(* Schneider Machine Expert - Basic project SHREDDER, file version 2.8.0.0 *)
(* ProjectInformations: Name=Mulino Bazzica *)
(* UserInformations: LastName=Dominici, FirstName=Erica, PhoneNumber=+39 0742 38501, Email=info@promas.com, Street=via XXV Aprile, 10/12, City=Trevi, ZipCode=06039, State=Perugia, Country=Italy *)

HARDWARE
  Cpu 0: TM221CE16T
  EthernetConfiguration: NetworkName=M221, IpAllocationMode=FixedAddress, IpAddress=192.168.0.230, SubnetMask=255.255.254.0
  SerialLineConfiguration: Baud=Baud19200, Parity=ParityEven, DataBits=DataBits8, StopBits=StopBits1, PhysicalMedium=PhysicalMediumRs485, TransmissionMode=TransmissionModeModbusRtu, SlaveId=1, Addressing=SlaveAddressing
  MastTask: UsePeriodScanMode=true, PeriodScan=100
  FastTask: Period=255
  CpuBehavior: StartingMode=StartInRun, AutoSaveRamOnEeprom=true, WatchdogPeriod=250

SYMBOLS  (address, symbol, comment, settings)
  %M0       KM_ALL_ON
  %M1       KM_M1_ON
  %M2       ALARM_KM1
  %M3       ALARM_QM1
  %M4       ALARM_EXTERNAL
  %MW0      FSM_RECYCLING
  %MW4      ALARMS
  %MW6      HMI_INP  "PLC INPUT STATUS"
  %MW7      HMI_OUT  "PLC OUTPUT STATUS"
  %MW8      HMI_CMD  "PLC COMMANDS"
  %MW10     MACHINE_STATE
  %MW18     BLOWER_TIME  "O0 - BLOWER ON"
  %MW19     BLOWER_DELAY_OFF  "O0 - BLOWER DELAY OFF TIME"
  %MW20     VALVES_TIME  "O1-VALVES_SWITCH"
  %TM0      TON_VALVES  [Base=OneSecond, IsDynamicPreset=true]
  %TM1      TON_M1  [Preset=10, Base=OneSecond, IsDynamicPreset=true]
  %TM2      M1_ALM_ON  [Preset=3, Base=OneSecond]
  %TM3      M1_ALM_OFF  [Preset=3, Base=OneSecond]
  %TM4      QM1_ALM_ON  [Preset=3, Base=OneSecond]
  %TM5      QM1_ALM_OFF  [Preset=3, Base=OneSecond]
  %TM6      TON_M1_OFF  [Preset=3, IsDynamicPreset=true]
  %TM7      MULINO_ALM_ON  [Preset=3, Base=OneSecond]
  %TM8      MULINO_ALM_OFF  [Preset=3, Base=OneSecond]
  %I0.0     FDBK_TERMICO_QM1  "MGNETOTERMICO QM1"
  %I0.1     CONTATTORE_KM1  "CONTATTORE KM1"
  %I0.2     START_BTN  "START"
  %I0.3     STOP_BTN  "STOP"
  %I0.4     GENERAL_ERR_MULINO  "ERRORE MULINO"
  %Q0.0     VALVE1_2  "VALVES 12"
  %Q0.1     SILO_2_P  "SOLO PICCOLO"
  %Q0.2     SILO_1_G  "SILO GRANDE"
  %Q0.6     CONTACTOR_ON  "FAN"

POU IN
  (* SectionNumber=1 *)

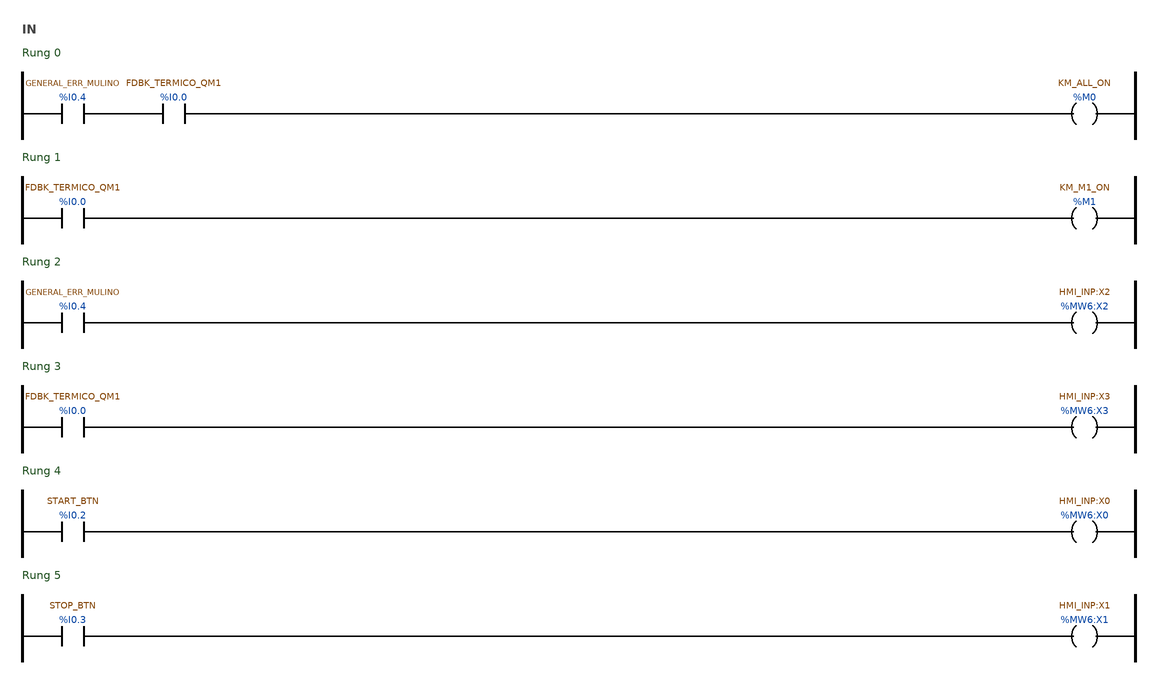

// Rung 0
  LD %I0.4                (* GENERAL_ERR_MULINO *)
  AND %I0.0               (* FDBK_TERMICO_QM1 *)
  ST %M0                  (* KM_ALL_ON *)
  // as ST:
  //   KM_ALL_ON := GENERAL_ERR_MULINO AND FDBK_TERMICO_QM1;

// Rung 1
  LD %I0.0                (* FDBK_TERMICO_QM1 *)
  ST %M1                  (* KM_M1_ON *)
  // as ST:
  //   KM_M1_ON := FDBK_TERMICO_QM1;

// Rung 2
  LD %I0.4                (* GENERAL_ERR_MULINO *)
  ST %MW6:X2              (* HMI_INP *)
  // as ST:
  //   HMI_INP:X2 := GENERAL_ERR_MULINO;

// Rung 3
  LD %I0.0                (* FDBK_TERMICO_QM1 *)
  ST %MW6:X3              (* HMI_INP *)
  // as ST:
  //   HMI_INP:X3 := FDBK_TERMICO_QM1;

// Rung 4
  LD %I0.2                (* START_BTN *)
  ST %MW6:X0              (* HMI_INP *)
  // as ST:
  //   HMI_INP:X0 := START_BTN;

// Rung 5
  LD %I0.3                (* STOP_BTN *)
  ST %MW6:X1              (* HMI_INP *)
  // as ST:
  //   HMI_INP:X1 := STOP_BTN;

POU FSM
  (* SectionNumber=2 *)

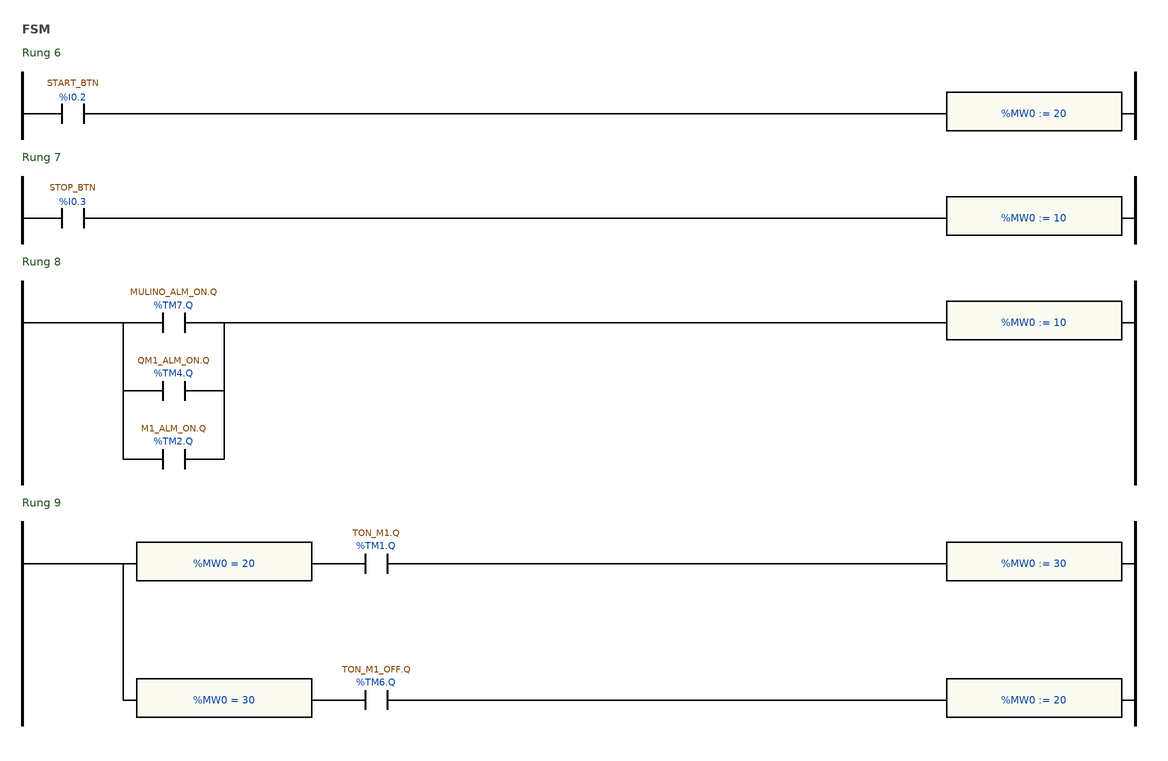

// Rung 6
  LD %I0.2                (* START_BTN *)
  [ %MW0 := 20 ]          (* FSM_RECYCLING *)
  // as ST:
  //   IF START_BTN THEN FSM_RECYCLING := 20; END_IF;

// Rung 7
  LD %I0.3                (* STOP_BTN *)
  [ %MW0 := 10 ]          (* FSM_RECYCLING *)
  // as ST:
  //   IF STOP_BTN THEN FSM_RECYCLING := 10; END_IF;

// Rung 8
  LD 1
  AND( %TM7.Q             (* MULINO_ALM_ON *)
  OR %TM4.Q               (* QM1_ALM_ON *)
  OR %TM2.Q               (* M1_ALM_ON *)
  )
  [ %MW0 := 10 ]          (* FSM_RECYCLING *)
  // as ST:
  //   IF MULINO_ALM_ON.Q OR QM1_ALM_ON.Q OR M1_ALM_ON.Q THEN FSM_RECYCLING := 10; END_IF;

// Rung 9
  LD 1
  MPS
  AND [ %MW0 = 20 ]       (* FSM_RECYCLING *)
  AND %TM1.Q              (* TON_M1 *)
  [ %MW0 := 30 ]          (* FSM_RECYCLING *)
  MPP
  AND [ %MW0 = 30 ]       (* FSM_RECYCLING *)
  AND %TM6.Q              (* TON_M1_OFF *)
  [ %MW0 := 20 ]          (* FSM_RECYCLING *)
  // as ST:
  //   IF FSM_RECYCLING = 20 AND TON_M1.Q THEN FSM_RECYCLING := 30; END_IF;
  //   IF FSM_RECYCLING = 30 AND TON_M1_OFF.Q THEN FSM_RECYCLING := 20; END_IF;

POU TIMERS
  (* SectionNumber=3 *)

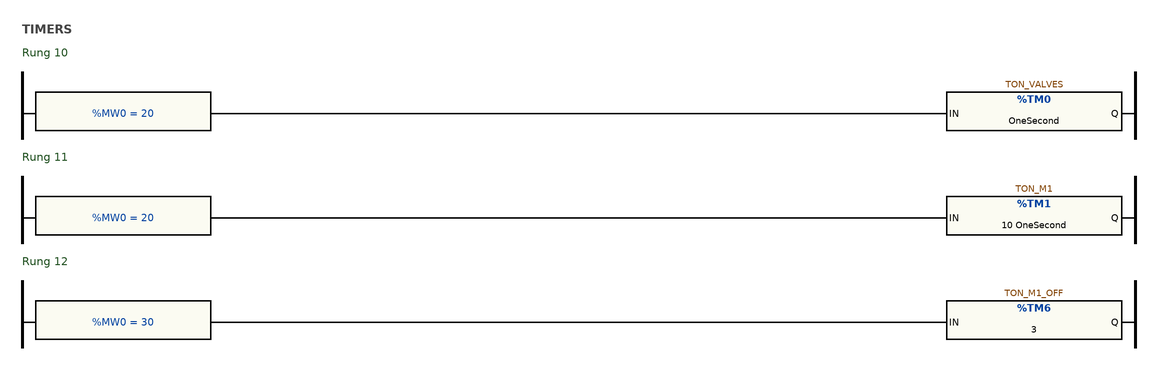

// Rung 10
  BLK %TM0                (* TON_VALVES *)
  LD [ %MW0 = 20 ]        (* FSM_RECYCLING *)
  IN
  END_BLK
  // as ST:
  //   TON_VALVES(IN := FSM_RECYCLING = 20);

// Rung 11
  BLK %TM1                (* TON_M1 *)
  LD [ %MW0 = 20 ]        (* FSM_RECYCLING *)
  IN
  END_BLK
  // as ST:
  //   TON_M1(IN := FSM_RECYCLING = 20);

// Rung 12
  BLK %TM6                (* TON_M1_OFF *)
  LD [ %MW0 = 30 ]        (* FSM_RECYCLING *)
  IN
  END_BLK
  // as ST:
  //   TON_M1_OFF(IN := FSM_RECYCLING = 30);

POU OUT
  (* SectionNumber=4 *)

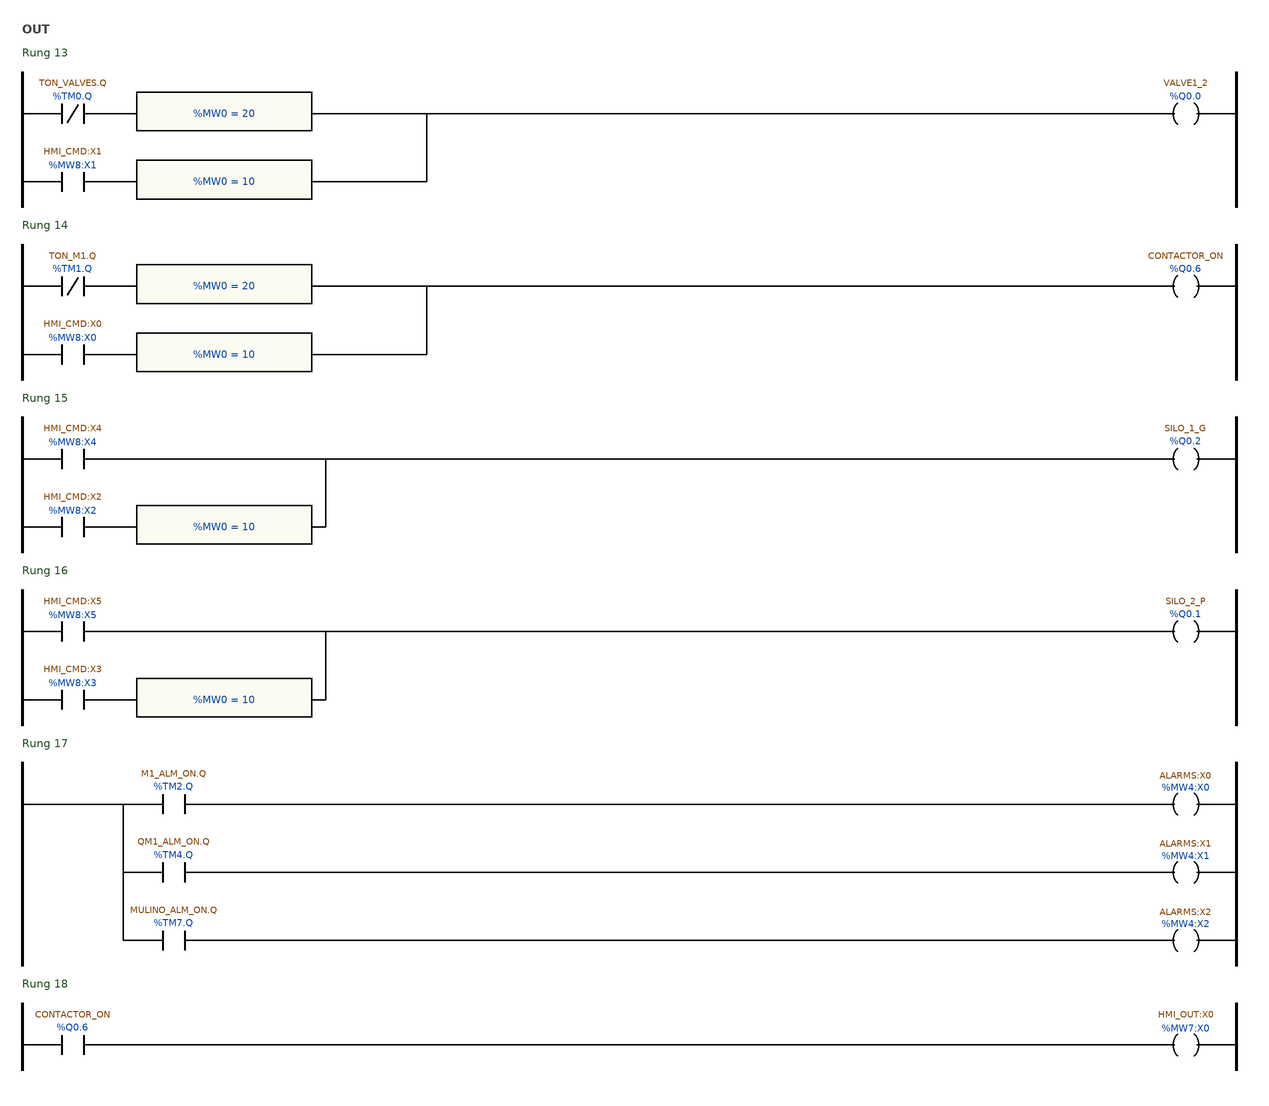

// Rung 13
  LDN %TM0.Q              (* TON_VALVES *)
  AND [ %MW0 = 20 ]       (* FSM_RECYCLING *)
  OR( %MW8:X1             (* HMI_CMD *)
  AND [ %MW0 = 10 ]       (* FSM_RECYCLING *)
  )
  ST %Q0.0                (* VALVE1_2 *)
  // as ST:
  //   VALVE1_2 := NOT TON_VALVES.Q AND FSM_RECYCLING = 20 OR HMI_CMD:X1 AND FSM_RECYCLING = 10;

// Rung 14
  LDN %TM1.Q              (* TON_M1 *)
  AND [ %MW0 = 20 ]       (* FSM_RECYCLING *)
  OR( %MW8:X0             (* HMI_CMD *)
  AND [ %MW0 = 10 ]       (* FSM_RECYCLING *)
  )
  ST %Q0.6                (* CONTACTOR_ON *)
  // as ST:
  //   CONTACTOR_ON := NOT TON_M1.Q AND FSM_RECYCLING = 20 OR HMI_CMD:X0 AND FSM_RECYCLING = 10;

// Rung 15
  LD %MW8:X4              (* HMI_CMD *)
  OR( %MW8:X2             (* HMI_CMD *)
  AND [ %MW0 = 10 ]       (* FSM_RECYCLING *)
  )
  ST %Q0.2                (* SILO_1_G *)
  // as ST:
  //   SILO_1_G := HMI_CMD:X4 OR HMI_CMD:X2 AND FSM_RECYCLING = 10;

// Rung 16
  LD %MW8:X5              (* HMI_CMD *)
  OR( %MW8:X3             (* HMI_CMD *)
  AND [ %MW0 = 10 ]       (* FSM_RECYCLING *)
  )
  ST %Q0.1                (* SILO_2_P *)
  // as ST:
  //   SILO_2_P := HMI_CMD:X5 OR HMI_CMD:X3 AND FSM_RECYCLING = 10;

// Rung 17
  LD 1
  MPS
  AND %TM2.Q              (* M1_ALM_ON *)
  ST %MW4:X0              (* ALARMS *)
  MRD
  AND %TM4.Q              (* QM1_ALM_ON *)
  ST %MW4:X1              (* ALARMS *)
  MPP
  AND %TM7.Q              (* MULINO_ALM_ON *)
  ST %MW4:X2              (* ALARMS *)
  // as ST:
  //   ALARMS:X0 := M1_ALM_ON.Q;
  //   ALARMS:X1 := QM1_ALM_ON.Q;
  //   ALARMS:X2 := MULINO_ALM_ON.Q;

// Rung 18
  LD %Q0.6                (* CONTACTOR_ON *)
  ST %MW7:X0              (* HMI_OUT *)
  // as ST:
  //   HMI_OUT:X0 := CONTACTOR_ON;

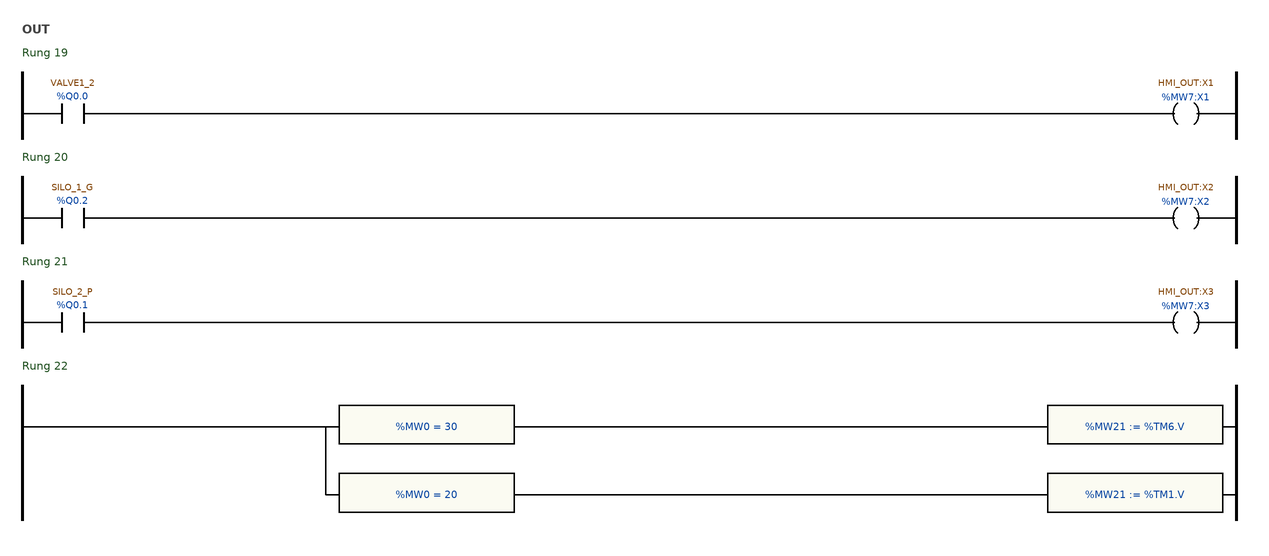

// Rung 19
  LD %Q0.0                (* VALVE1_2 *)
  ST %MW7:X1              (* HMI_OUT *)
  // as ST:
  //   HMI_OUT:X1 := VALVE1_2;

// Rung 20
  LD %Q0.2                (* SILO_1_G *)
  ST %MW7:X2              (* HMI_OUT *)
  // as ST:
  //   HMI_OUT:X2 := SILO_1_G;

// Rung 21
  LD %Q0.1                (* SILO_2_P *)
  ST %MW7:X3              (* HMI_OUT *)
  // as ST:
  //   HMI_OUT:X3 := SILO_2_P;

// Rung 22
  LD 1
  MPS
  AND [ %MW0 = 30 ]       (* FSM_RECYCLING *)
  [ %MW21 := %TM6.V ]     (* TON_M1_OFF *)
  MPP
  AND [ %MW0 = 20 ]       (* FSM_RECYCLING *)
  [ %MW21 := %TM1.V ]     (* TON_M1 *)
  // as ST:
  //   IF FSM_RECYCLING = 30 THEN %MW21 := TON_M1_OFF.V; END_IF;
  //   IF FSM_RECYCLING = 20 THEN %MW21 := TON_M1.V; END_IF;

POU SETTINGS
  (* SectionNumber=5 *)

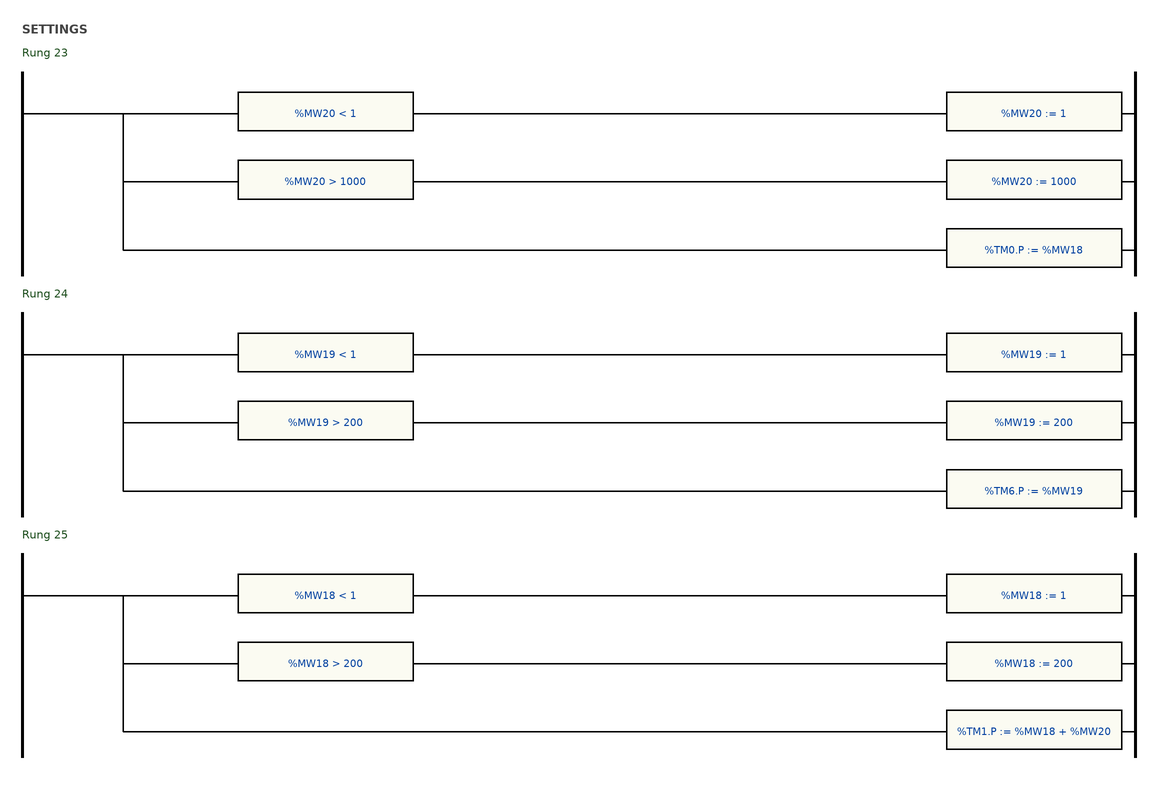

// Rung 23
  LD 1
  MPS
  AND [ %MW20 < 1 ]       (* VALVES_TIME *)
  [ %MW20 := 1 ]          (* VALVES_TIME *)
  MRD
  AND [ %MW20 > 1000 ]    (* VALVES_TIME *)
  [ %MW20 := 1000 ]       (* VALVES_TIME *)
  MPP
  [ %TM0.P := %MW18 ]     (* TON_VALVES, BLOWER_TIME *)
  // as ST:
  //   IF VALVES_TIME < 1 THEN VALVES_TIME := 1; END_IF;
  //   IF VALVES_TIME > 1000 THEN VALVES_TIME := 1000; END_IF;
  //   TON_VALVES.P := BLOWER_TIME;

// Rung 24
  LD 1
  MPS
  AND [ %MW19 < 1 ]       (* BLOWER_DELAY_OFF *)
  [ %MW19 := 1 ]          (* BLOWER_DELAY_OFF *)
  MRD
  AND [ %MW19 > 200 ]     (* BLOWER_DELAY_OFF *)
  [ %MW19 := 200 ]        (* BLOWER_DELAY_OFF *)
  MPP
  [ %TM6.P := %MW19 ]     (* TON_M1_OFF, BLOWER_DELAY_OFF *)
  // as ST:
  //   IF BLOWER_DELAY_OFF < 1 THEN BLOWER_DELAY_OFF := 1; END_IF;
  //   IF BLOWER_DELAY_OFF > 200 THEN BLOWER_DELAY_OFF := 200; END_IF;
  //   TON_M1_OFF.P := BLOWER_DELAY_OFF;

// Rung 25
  LD 1
  MPS
  AND [ %MW18 < 1 ]       (* BLOWER_TIME *)
  [ %MW18 := 1 ]          (* BLOWER_TIME *)
  MRD
  AND [ %MW18 > 200 ]     (* BLOWER_TIME *)
  [ %MW18 := 200 ]        (* BLOWER_TIME *)
  MPP
  [ %TM1.P := %MW18 + %MW20 ](* TON_M1, BLOWER_TIME, VALVES_TIME *)
  // as ST:
  //   IF BLOWER_TIME < 1 THEN BLOWER_TIME := 1; END_IF;
  //   IF BLOWER_TIME > 200 THEN BLOWER_TIME := 200; END_IF;
  //   TON_M1.P := BLOWER_TIME + VALVES_TIME;

POU ALARMS
  (* SectionNumber=6 *)

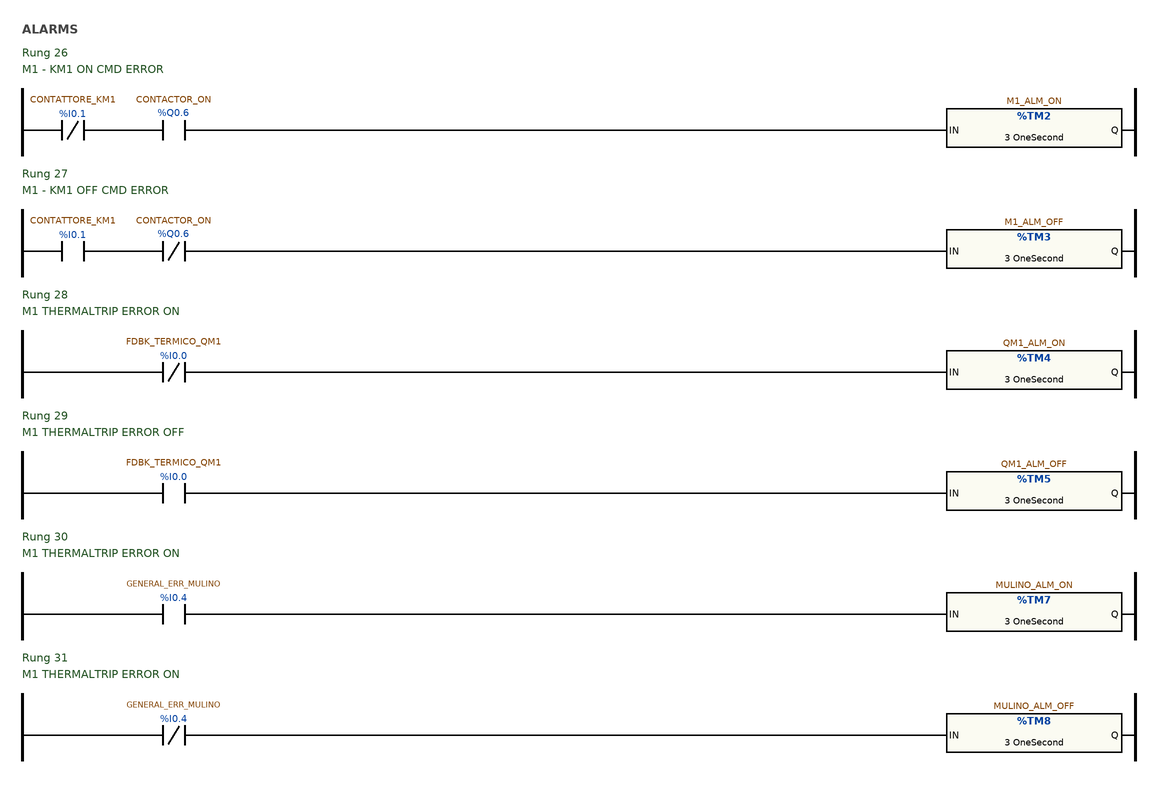

// Rung 26
// M1 - KM1 ON CMD ERROR
  BLK %TM2                (* M1_ALM_ON *)
  LDN %I0.1               (* CONTATTORE_KM1 *)
  AND %Q0.6               (* CONTACTOR_ON *)
  IN
  END_BLK
  // as ST:
  //   M1_ALM_ON(IN := NOT CONTATTORE_KM1 AND CONTACTOR_ON);

// Rung 27
// M1 - KM1 OFF CMD ERROR
  BLK %TM3                (* M1_ALM_OFF *)
  LD %I0.1                (* CONTATTORE_KM1 *)
  ANDN %Q0.6              (* CONTACTOR_ON *)
  IN
  END_BLK
  // as ST:
  //   M1_ALM_OFF(IN := CONTATTORE_KM1 AND NOT CONTACTOR_ON);

// Rung 28
// M1 THERMALTRIP ERROR ON
  BLK %TM4                (* QM1_ALM_ON *)
  LDN %I0.0               (* FDBK_TERMICO_QM1 *)
  IN
  END_BLK
  // as ST:
  //   QM1_ALM_ON(IN := NOT FDBK_TERMICO_QM1);

// Rung 29
// M1 THERMALTRIP ERROR OFF
  BLK %TM5                (* QM1_ALM_OFF *)
  LD %I0.0                (* FDBK_TERMICO_QM1 *)
  IN
  END_BLK
  // as ST:
  //   QM1_ALM_OFF(IN := FDBK_TERMICO_QM1);

// Rung 30
// M1 THERMALTRIP ERROR ON
  BLK %TM7                (* MULINO_ALM_ON *)
  LD %I0.4                (* GENERAL_ERR_MULINO *)
  IN
  END_BLK
  // as ST:
  //   MULINO_ALM_ON(IN := GENERAL_ERR_MULINO);

// Rung 31
// M1 THERMALTRIP ERROR ON
  BLK %TM8                (* MULINO_ALM_OFF *)
  LDN %I0.4               (* GENERAL_ERR_MULINO *)
  IN
  END_BLK
  // as ST:
  //   MULINO_ALM_OFF(IN := NOT GENERAL_ERR_MULINO);

POU CONNECTION
  (* SectionNumber=7 *)

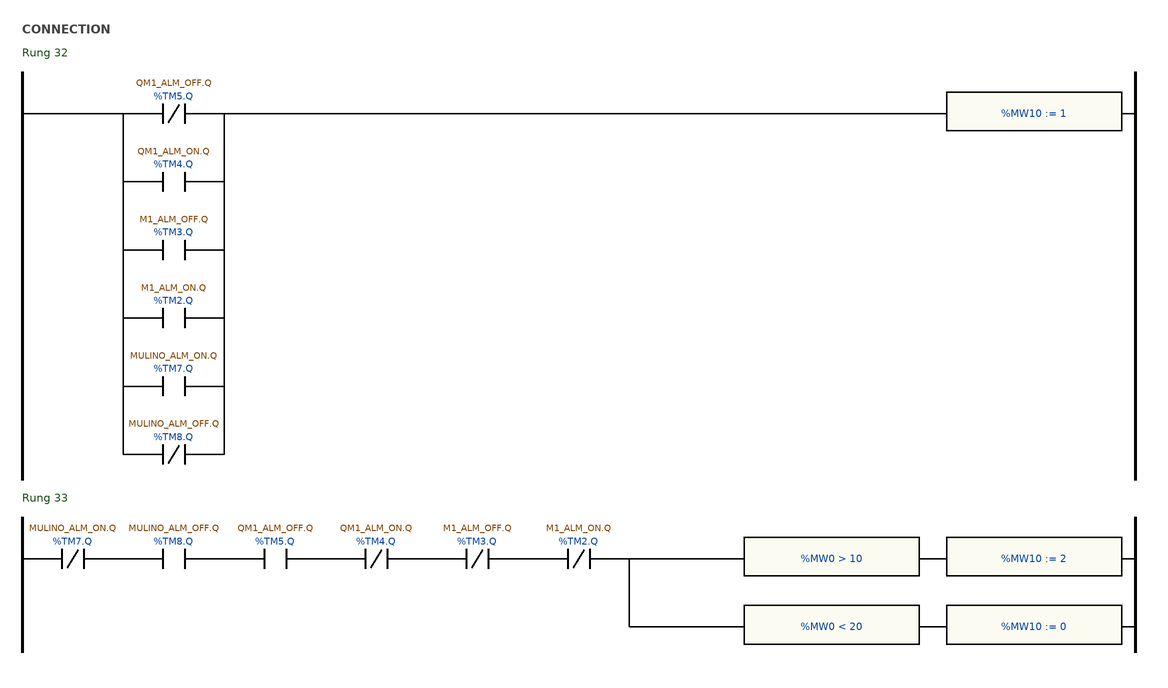

// Rung 32
  LD 1
  AND(N %TM5.Q            (* QM1_ALM_OFF *)
  OR %TM4.Q               (* QM1_ALM_ON *)
  OR %TM3.Q               (* M1_ALM_OFF *)
  OR %TM2.Q               (* M1_ALM_ON *)
  OR %TM7.Q               (* MULINO_ALM_ON *)
  ORN %TM8.Q              (* MULINO_ALM_OFF *)
  )
  [ %MW10 := 1 ]          (* MACHINE_STATE *)
  // as ST:
  //   IF NOT QM1_ALM_OFF.Q OR QM1_ALM_ON.Q OR M1_ALM_OFF.Q OR M1_ALM_ON.Q OR MULINO_ALM_ON.Q OR NOT MULINO_ALM_OFF.Q THEN MACHINE_STATE := 1; END_IF;

// Rung 33
  LDN %TM7.Q              (* MULINO_ALM_ON *)
  AND %TM8.Q              (* MULINO_ALM_OFF *)
  AND %TM5.Q              (* QM1_ALM_OFF *)
  ANDN %TM4.Q             (* QM1_ALM_ON *)
  ANDN %TM3.Q             (* M1_ALM_OFF *)
  ANDN %TM2.Q             (* M1_ALM_ON *)
  MPS
  AND [ %MW0 > 10 ]       (* FSM_RECYCLING *)
  [ %MW10 := 2 ]          (* MACHINE_STATE *)
  MPP
  AND [ %MW0 < 20 ]       (* FSM_RECYCLING *)
  [ %MW10 := 0 ]          (* MACHINE_STATE *)
  // as ST:
  //   IF NOT MULINO_ALM_ON.Q AND MULINO_ALM_OFF.Q AND QM1_ALM_OFF.Q AND NOT QM1_ALM_ON.Q AND NOT M1_ALM_OFF.Q AND NOT M1_ALM_ON.Q AND FSM_RECYCLING > 10 THEN MACHINE_STATE := 2; END_IF;
  //   IF NOT MULINO_ALM_ON.Q AND MULINO_ALM_OFF.Q AND QM1_ALM_OFF.Q AND NOT QM1_ALM_ON.Q AND NOT M1_ALM_OFF.Q AND NOT M1_ALM_ON.Q AND FSM_RECYCLING < 20 THEN MACHINE_STATE := 0; END_IF;
